Fanuc TP program (LS listing): up202.ls

/PROG  UP202
/ATTR
OWNER		= AUROM;
COMMENT		= "Camb. Herr. SP1";
PROG_SIZE	= 1902;
CREATE		= DATE 03-15-00  TIME 13:37:40;
MODIFIED	= DATE 16-11-30  TIME 02:42:42;
FILE_NAME	= ;
VERSION		= 0;
LINE_COUNT	= 7;
MEMORY_SIZE	= 3254;
PROTECT		= READ_WRITE;
TCD:  STACK_SIZE	= 500,
      TASK_PRIORITY	= 50,
      TIME_SLICE	= 0,
      BUSY_LAMP_OFF	= 0,
      ABORT_REQUEST	= 0,
      PAUSE_REQUEST	= 0;
DEFAULT_GROUP	= 1,1,1,1,*;
CONTROL_CODE	= 00000000 00000000;
/MN
   1:  UTOOL_NUM=1 ;
   2:  UFRAME_NUM=0 ;
   3:  PAYLOAD[1] ;
   4:J P[1] 100% CNT0 ACC100 TB    .10sec,P-SPS    ;
      1:  TC_ONLINE (ON) ;
      2:  DO[23]=OFF ;
      3:  CALL MAKRO050    ;
      4:  !Lib. de Herramientas ;
      5:  DO[80]=ON ;
      6:  DO[78]=OFF ;
      7:  DO[77]=ON ;
      8:  DO[75]=OFF ;
      9:  !Lib. de Anticolisiones ;
     10:  DO[41]=ON ;
     11:  DO[42]=ON ;
     12:  DO[43]=ON ;
     13:  DO[44]=ON ;
     14:  !Apagar Pos. Base ;
     15:  DO[15]=OFF ;
     16:  !Robot en Trayectoria ;
     17:  DO[16]=ON ;
     18:  WAIT (DI[23])    ;
     19:  DO[23]=ON ;
     20:  TC_ONLINE (M[2] AND M[30] AND M[31] AND M[33] AND M[95] AND M[96]) ;
       ------ ;
   5:  !Cambio de Herramienta ;
   6:J P[2] 100% CNT0 ACC100 TB    .10sec,P-SPS    ;
      1:  TC_ONLINE (ON) ;
      2:  DO[23]=OFF ;
      3:  DO[17]=ON ;
      4:  GO[19]=(11) ;
      5:  WAIT (DI[17])    ;
      6:  DO[17]=OFF ;
      7:  GO[19]=(0) ;
      8:  WAIT (DI[23])    ;
      9:  DO[23]=ON ;
     10:  TC_ONLINE (M[2] AND M[30] AND M[31] AND M[33] AND M[95] AND M[96]) ;
       ------ ;
   7:J P[3] 100% CNT0 ACC100 TB    .10sec,P-SPS    ;
      1:  TC_ONLINE (ON) ;
      2:  DO[23]=OFF ;
      3:  WAIT (DI[23])    ;
      4:  DO[23]=ON ;
      5:  TC_ONLINE (M[2] AND M[30] AND M[31] AND M[33] AND M[95] AND M[96]) ;
       ------ ;
/POS
P[1]{
   GP1:
	UF : 0, UT : 1,		CONFIG : 'N U T, 0, 0, 0',
	X =  -464.787  mm,	Y =  -676.745  mm,	Z =  1035.419  mm,
	W =   142.550 deg,	P =    72.302 deg,	R =  -130.575 deg
   GP2:
	UF : 0, UT : 1,
	J1=   100.000  mm
   GP3:
	UF : 0, UT : 1,
	J1=     0.000  mm
   GP4:
	UF : 0, UT : 1,
	J1=     0.000  mm
};
P[2]{
   GP1:
	UF : 0, UT : 1,		CONFIG : 'N U T, 0, 0, 0',
	X =  -464.787  mm,	Y =  -676.745  mm,	Z =  1035.419  mm,
	W =   142.550 deg,	P =    72.302 deg,	R =  -130.575 deg
   GP2:
	UF : 0, UT : 1,
	J1=   100.000  mm
   GP3:
	UF : 0, UT : 1,
	J1=     0.000  mm
   GP4:
	UF : 0, UT : 1,
	J1=     0.000  mm
};
P[3]{
   GP1:
	UF : 0, UT : 1,		CONFIG : 'N U T, 0, 0, 0',
	X =  -464.787  mm,	Y =  -676.745  mm,	Z =  1035.419  mm,
	W =   142.550 deg,	P =    72.302 deg,	R =  -130.575 deg
   GP2:
	UF : 0, UT : 1,
	J1=   100.000  mm
   GP3:
	UF : 0, UT : 1,
	J1=     0.000  mm
   GP4:
	UF : 0, UT : 1,
	J1=     0.000  mm
};
/END
